PROGRAM MAIN
VAR
END_VAR

Runtime();

JobsExample();
StatesExample();

END_PROGRAM

(* stored: Version 1.1.0.1
   POU MAIN: Id {a2fd94c7-ef89-4407-b170-226415532fd6}, SpecialFunc None *)
